// TwinCAT 3 PLC project ZeroSpanCalibration
// ProgramVersion: 3.1.4023.0
// libraries:
//   Tc2_Standard, * (Beckhoff Automation GmbH)
//   Tc2_System, * (Beckhoff Automation GmbH)
//   Tc3_Module, * (Beckhoff Automation GmbH)
// project tree:
//   / PlcTask.TcTTO
//   POUs/ FB_ZeroSpanCalibration.TcPOU, GVL_ZeroSpanCalibration.TcGVL, MAIN.TcPOU
// real-time tasks:
//   TASK PlcTask: cycle T#10ms, priority 20, ADS port 350

CONFIGURATION ZeroSpanCalibration
    RESOURCE PLC ON TwinCAT3
        TASK PlcTask(INTERVAL := T#10ms, PRIORITY := 20);
        PROGRAM MAIN WITH PlcTask : MAIN;
    END_RESOURCE
END_CONFIGURATION

// ---- POUs/GVL_ZeroSpanCalibration.TcGVL
VAR_GLOBAL CONSTANT
	nInitialize: SINT := 0;
	nStep: SINT := 1;
END_VAR

// ---- POUs/MAIN.TcPOU
PROGRAM MAIN
VAR
END_VAR

END_PROGRAM

// ---- POUs/FB_ZeroSpanCalibration.TcPOU
FUNCTION_BLOCK FB_ZeroSpanCalibration
VAR_INPUT
	nMethodType: SINT;	//Method tpye: '0' for initialization, '1' for start-up
	fIn: LREAL;			//Instrument input. e.g. sensor input, valve input
END_VAR
VAR_OUTPUT	
	f_y1y2: LREAL;		//If the signal is rising then zero error (y1). If the signal is falling then span error (y2).
END_VAR
VAR
	rtb_TSamp: LREAL;
	rtb_Diff: LREAL;
	rtb_Compare: BOOL;
	rtb_Compare_o: BOOL;
	UD_DSTATE: LREAL;
	DelayInput1_DSTATE: BOOL;
	DelayInput1_DSTATE_a: BOOL;
END_VAR

CASE nMethodType OF
    nInitialize: 
        // Initialize conditions for unit delay   
        UD_DSTATE := 0.0;
        DelayInput1_DSTATE := FALSE;
        DelayInput1_DSTATE_a := FALSE;        
        // Initialize condition for the system output
        f_y1y2 := 0.0;      
    nStep:       
        //y = u * K where K = 1 / ( w * Ts ) *)
        rtb_TSamp := fIn * 20.0;       
        rtb_Diff := rtb_TSamp - UD_DSTATE;   
        rtb_Compare := rtb_Diff > 0.0;      
        rtb_Compare_o := rtb_Diff < 0.0;        

        IF UDINT_TO_DINT(BOOL_TO_UDINT(BOOL_TO_DINT(rtb_Compare) > BOOL_TO_DINT(DelayInput1_DSTATE)) + BOOL_TO_UDINT(BOOL_TO_DINT(rtb_Compare_o) > BOOL_TO_DINT(DelayInput1_DSTATE_a))) = 1 THEN 
        	f_y1y2 := fIn;           
        END_IF;
        UD_DSTATE := rtb_TSamp;   
        DelayInput1_DSTATE := rtb_Compare;
        DelayInput1_DSTATE_a := rtb_Compare_o;
END_CASE;

END_FUNCTION_BLOCK
